// TIA Portal V19 export
DATA_BLOCK "IPC_Send_Buffer_Log_MACCHINA"   // DB190
// stored: MemoryReserve 100
   VAR RETAIN
      lastId : DInt;
      msg : Array[1.."LOG_MSG_ITEMS"] of "IPC_Msg_Generico";
   END_VAR
BEGIN
END_DATA_BLOCK
